// TIA Portal V20 export
// export: Created 2025-12-01T14:57:19.7177063Z, ExportSetting None, DisplayName Totally Integrated Automation Portal, DisplayVersion V20 Update 3, DisplayName TIA Portal Openness, DisplayVersion V20 Update 3, DisplayName TIA Portal Version Control Interface, DisplayVersion V20 Update 3, DisplayName STEP 7 Professional, DisplayVersion V20 Update 3, DisplayName STEP 7 Safety, DisplayVersion V20 Update 2, DisplayName WinCC Basic/Comfort/Advanced, DisplayVersion V20 Update 3, DisplayName WinCC Professional, DisplayVersion V20 Update 3, DisplayName WinCC Unified, DisplayVersion V20 Update 3
DATA_BLOCK "DB301_Velocidad_FSS"   // DB301
{ S7_Optimized_Access := 'FALSE' }
// stored: AutoNumber false
   VAR RETAIN
      carga : Struct
         Rapida : Int := 24000;
         Media : Int := 15000;
         Lenta : Int := 15000;
         Posicionado : Int := 2500;
      END_STRUCT;
      Descarga : Struct
         Rapida : Int := 24000;
         Media : Int := 15000;
         Lenta : Int := 15000;
         Posicionado : Int := 2500;
      END_STRUCT;
   END_VAR
BEGIN
END_DATA_BLOCK
